INTERFACE I_Cycle EXTENDS I_Object

METHOD PUBLIC M_Call
VAR_INPUT
END_VAR
END_METHOD

END_INTERFACE

(* stored: Version 1.1.0.1
   Itf I_Cycle: Id {e1e2ff06-3bf6-45ba-91e5-14895b5625fb}
   Method M_Call: Id {34b9e3de-1b13-0ba0-374d-6aeb7f2678a3} *)
